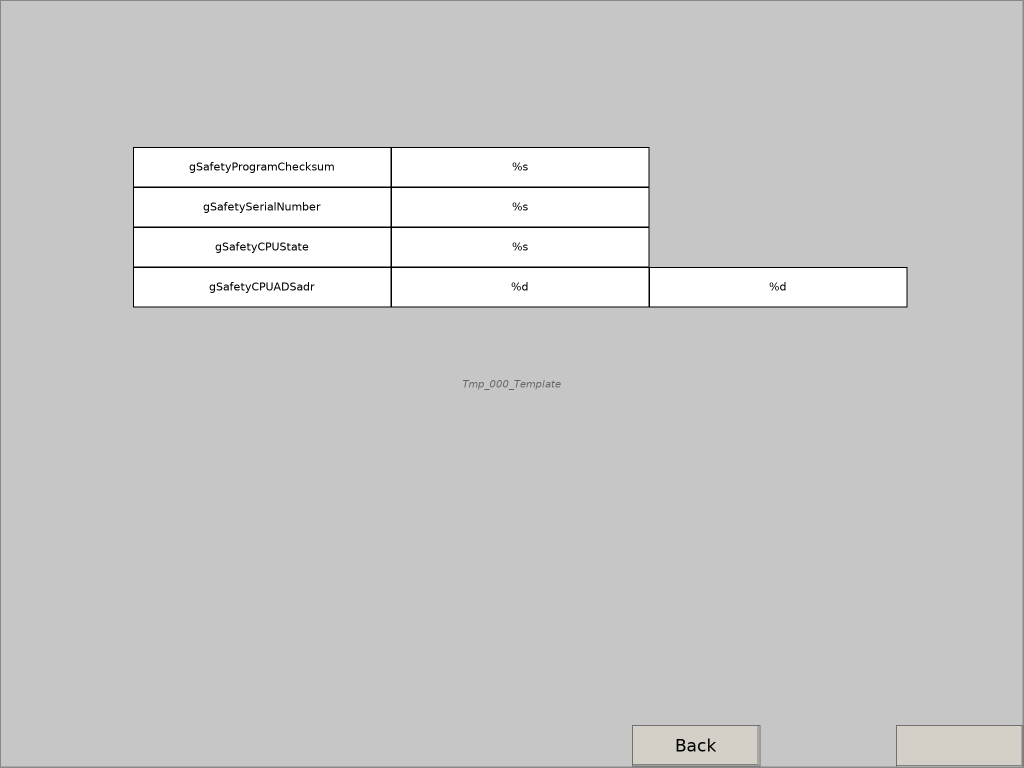
VISUALIZATION Saf_701_SafetyChecksum  // 1024x768
    Frame (0,0 1024x768)
        shows Tmp_000_Template(header := gHMIData.hmiHeader)
    Rectangle (1226,468 2x0)
    Rectangle (133,147 258x40), "gSafetyProgramChecksum"
    Rectangle (133,187 258x40), "gSafetySerialNumber"
    Rectangle (133,227 258x40), "gSafetyCPUState"
    Rectangle (133,267 258x40), "gSafetyCPUADSadr"
    Rectangle (391,147 258x40), "%s", text variable: Safety.gSafetyProgramChecksum, text list: ''
    Rectangle (391,187 258x40), "%s", text variable: Safety.gSafetySerialNumber
    Rectangle (391,227 258x40), "%s", text variable: Safety.gSafetyCPUState
    Rectangle (391,267 258x40), "%d", text variable: Safety.gSafetyCPUADSadr.netId
    Rectangle (649,267 258x40), "%d", text variable: Safety.gSafetyCPUADSadr.port
    Button (632,725 128x41), "Back"
        OnMouseClick: change screen: Saf_700_SafetyStatus
    Button (896,725 128x42)
END_VISUALIZATION

(* stored: Version 1.1.0.1, ProductVersion 3.1.4024.12
   Visu Saf_701_SafetyChecksum: Id {c564314e-c6da-4230-838d-e7e21aebfb47} *)
